(* Schneider Machine Expert - Basic project Exercise-10 - Multiple Motor Connections with using Memory Bits, file version 2.9.0.0 *)
(* ProjectInformations: Name=New project *)

HARDWARE
  Cpu 0: TM221CE24R
  EthernetConfiguration: NetworkName=M221, IpAllocationMode=FixedAddress, IpAddress=0.0.0.0, SubnetMask=0.0.0.0
  SerialLineConfiguration: Baud=Baud19200, Parity=ParityEven, DataBits=DataBits8, StopBits=StopBits1, PhysicalMedium=PhysicalMediumRs485, SlaveId=1, Addressing=SlaveAddressing
  MastTask: UsePeriodScanMode=false, PeriodScan=100
  FastTask: Period=255
  CpuBehavior: StartingMode=StartAsPreviousState, AutoSaveRamOnEeprom=true, WatchdogPeriod=250

SYMBOLS  (address, symbol, comment, settings)
  %M0       MEMORY_BIT
  %I0.0     SWITCH_1
  %Q0.0     MOTOR_1
  %Q0.1     MOTOR_2
  %Q0.2     MOTOR_3
  %Q0.3     MOTOR_4

POU New POU
  (* SectionNumber=1 *)

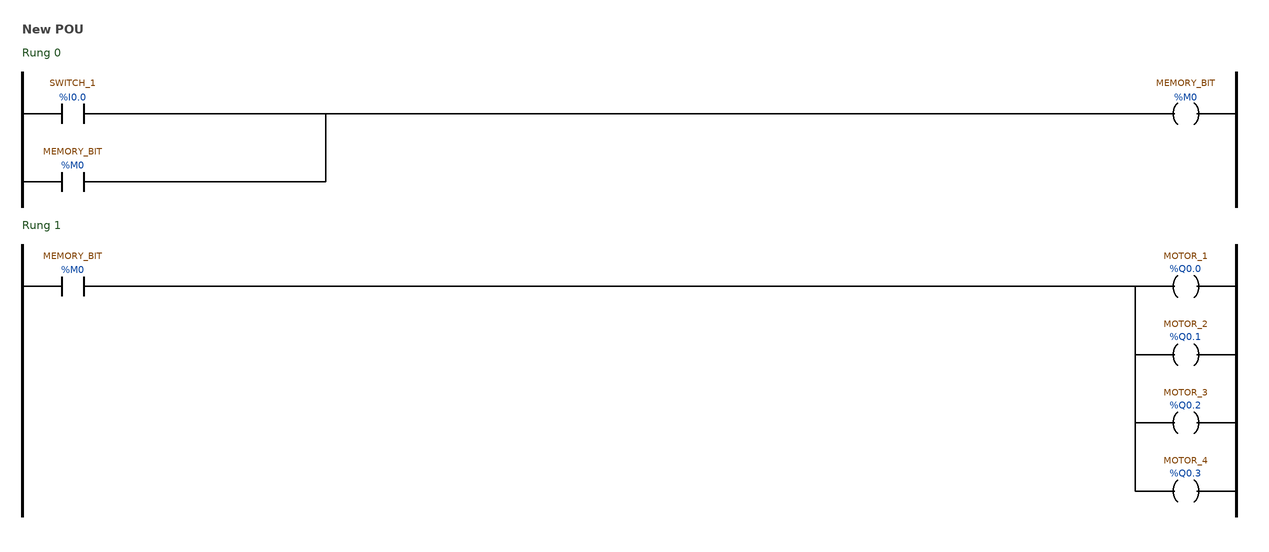

// Rung 0
  LD %I0.0                (* SWITCH_1 *)
  OR %M0                  (* MEMORY_BIT *)
  ST %M0                  (* MEMORY_BIT *)
  // as ST:
  //   MEMORY_BIT := SWITCH_1 OR MEMORY_BIT;

// Rung 1
  LD %M0                  (* MEMORY_BIT *)
  ST %Q0.0                (* MOTOR_1 *)
  ST %Q0.1                (* MOTOR_2 *)
  ST %Q0.2                (* MOTOR_3 *)
  ST %Q0.3                (* MOTOR_4 *)
  // as ST:
  //   MOTOR_1 := MEMORY_BIT;
  //   MOTOR_2 := MEMORY_BIT;
  //   MOTOR_3 := MEMORY_BIT;
  //   MOTOR_4 := MEMORY_BIT;
